// TIA Portal project "2020-10-23_StartStopMotoreNA-NC" (V16)

(* hardware
DEVICE "S7-1200 station_1"  S7-1200 Station
   slot 0: "Telaio di montaggio_0"  Rack  V1.0
   slot 1: "PLC_1"  CPU 1215C DC/DC/DC  6ES7 215-1AG40-0XB0  V4.2
*)

// ===== PLC "PLC_1"  CPU 1215C DC/DC/DC =====

VAR_GLOBAL   // PLC tag table "Tabella delle variabili standard"
   "Vent_A_NA" AT %I0.0 : Bool;
   "Vent_B_NC" AT %I0.1 : Bool;
   "Vent_C_NA" AT %I0.2 : Bool;
   "Start_NA" AT %I0.3 : Bool;
   "Stop_NC" AT %I0.4 : Bool;
   "Allarme_NC" AT %I0.5 : Bool;
   "Ripristino_NA" AT %I0.6 : Bool;
   "In7" AT %I0.7 : Bool;
   "Motore" AT %Q0.0 : Bool;
   "Vent_2su3_OK" AT %Q0.1 : Bool;
   "Allarme_mem" AT %M6.1 : Bool;
   "M_IB0_NCNA" AT %MB0 : Byte;   // indica tutte le variabili di memoria da 0.0 a 0.7
   "Vent_A" AT %M0.0 : Bool;
   "Vent_B" AT %M0.1 : Bool;
   "Vent_C" AT %M0.2 : Bool;
   "Start" AT %M0.3 : Bool;
   "Stop" AT %M0.4 : Bool;
   "Allarme" AT %M0.5 : Bool;
   "Ripristino" AT %M0.6 : Bool;
   "Sempre_vera" AT %M6.0 : Bool;
   "Ingressi" AT %IB0 : Byte;   // indica tutti gli ingressi da 0.0 a 0.7
   "XXX_Start_old" AT %M1.3 : Bool;
   "XXX_Ripristino_old" AT %M1.6 : Bool;
END_VAR

VAR_GLOBAL CONSTANT   // PLC tag table "Tabella delle variabili standard"
   "Maschera NCNA" : Byte := 2#00110010;
END_VAR

ORGANIZATION_BLOCK "Main"   // OB1, LAD, ProgramCycle
TITLE = "Main Program Sweep (Cycle)"
{ S7_Optimized_Access := 'TRUE' }
VERSION : 0.1
// Gestione di un motore, con almeno 2 ventilatori su 3 che funzionano e un allarme con memorizzazione ripristino e rientro
// 
// Gestione Maschera e rilevatori di fronte
// 
// I0.0, Vent_A, NA
// I0.1, Vent_B, NC
// I0.2, Vent_C, NA
// I0.3, Start, NA
// I0.4, Stop, NC
// I0.5 Allarme, NC
// I0.6 Ripristino, NA
// 
// Q0.0 Motore
// Q0.1 Ventilazione OK (almeno 2 ventilatori su 3 sono in funzione)
// 
// M0.0 Allarme memorizzato (Lampada di allarme)
   VAR_TEMP   // added for the SCL form of the ladder/FBD networks
      _w1 : Bool;
   END_VAR
BEGIN

REGION Network 1: Bit Sempre_vero
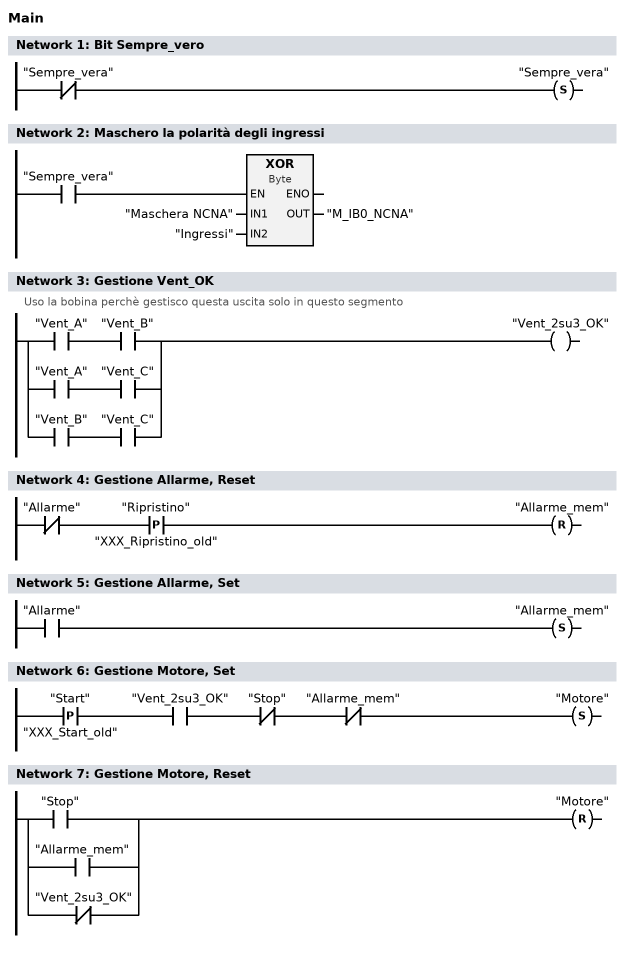
   RUNG wire#powerrail
      I_Contact( "Sempre_vera" )
      S_Coil( "Sempre_vera" )
   END_RUNG
   // the same network as SCL:
   IF NOT "Sempre_vera" THEN "Sempre_vera" := TRUE; END_IF;
END_REGION

REGION Network 2: Maschero la polarità degli ingressi
   IF "Sempre_vera" THEN "M_IB0_NCNA" := "Maschera NCNA" XOR "Ingressi"; END_IF;
END_REGION

REGION Network 3: Gestione Vent_OK
   // Uso la bobina perchè gestisco questa uscita solo in questo segmento
   RUNG wire#powerrail
      Contact( "Vent_A" )
      Contact( "Vent_B" )
      wire#w1
      Coil( "Vent_2su3_OK" )
   END_RUNG
   RUNG wire#powerrail
      Contact( "Vent_A" )
      Contact( "Vent_C" )
   END_RUNG wire#w1
   RUNG wire#powerrail
      Contact( "Vent_B" )
      Contact( "Vent_C" )
   END_RUNG wire#w1
   // the same network as SCL:
   "Vent_2su3_OK" := ("Vent_A" AND "Vent_B") OR ("Vent_A" AND "Vent_C") OR ("Vent_B" AND "Vent_C");
END_REGION

REGION Network 4: Gestione Allarme, Reset
   RUNG wire#powerrail
      I_Contact( "Allarme" )
      P_Contact(operand := "Ripristino", bit := "XXX_Ripristino_old")
      R_Coil( "Allarme_mem" )
   END_RUNG
   // the same network as SCL:
   #_w1 := NOT "Allarme" AND "Ripristino" AND NOT "XXX_Ripristino_old";   // rising edge of "Ripristino"
   "XXX_Ripristino_old" := "Ripristino";
   IF #_w1 THEN "Allarme_mem" := FALSE; END_IF;
END_REGION

REGION Network 5: Gestione Allarme, Set
   RUNG wire#powerrail
      Contact( "Allarme" )
      S_Coil( "Allarme_mem" )
   END_RUNG
   // the same network as SCL:
   IF "Allarme" THEN "Allarme_mem" := TRUE; END_IF;
END_REGION

REGION Network 6: Gestione Motore, Set
   RUNG wire#powerrail
      P_Contact(operand := "Start", bit := "XXX_Start_old")
      Contact( "Vent_2su3_OK" )
      I_Contact( "Stop" )
      I_Contact( "Allarme_mem" )
      S_Coil( "Motore" )
   END_RUNG
   // the same network as SCL:
   #_w1 := "Start" AND NOT "XXX_Start_old";   // rising edge of "Start"
   "XXX_Start_old" := "Start";
   IF #_w1 AND "Vent_2su3_OK" AND NOT "Stop" AND NOT "Allarme_mem" THEN "Motore" := TRUE; END_IF;
END_REGION

REGION Network 7: Gestione Motore, Reset
   RUNG wire#powerrail
      Contact( "Stop" )
      wire#w1
      R_Coil( "Motore" )
   END_RUNG
   RUNG wire#powerrail
      Contact( "Allarme_mem" )
   END_RUNG wire#w1
   RUNG wire#powerrail
      I_Contact( "Vent_2su3_OK" )
   END_RUNG wire#w1
   // the same network as SCL:
   IF "Stop" OR "Allarme_mem" OR NOT "Vent_2su3_OK" THEN "Motore" := FALSE; END_IF;
END_REGION
END_ORGANIZATION_BLOCK